// SIMATIC S7-200 project (STEP 7-Micro/WIN), CPU 224XP CN REL 02.01

ORGANIZATION_BLOCK 主程序:OB1
TITLE=程序注释；自由口通讯（甲机通过自由口通讯控制乙机电机）
BEGIN
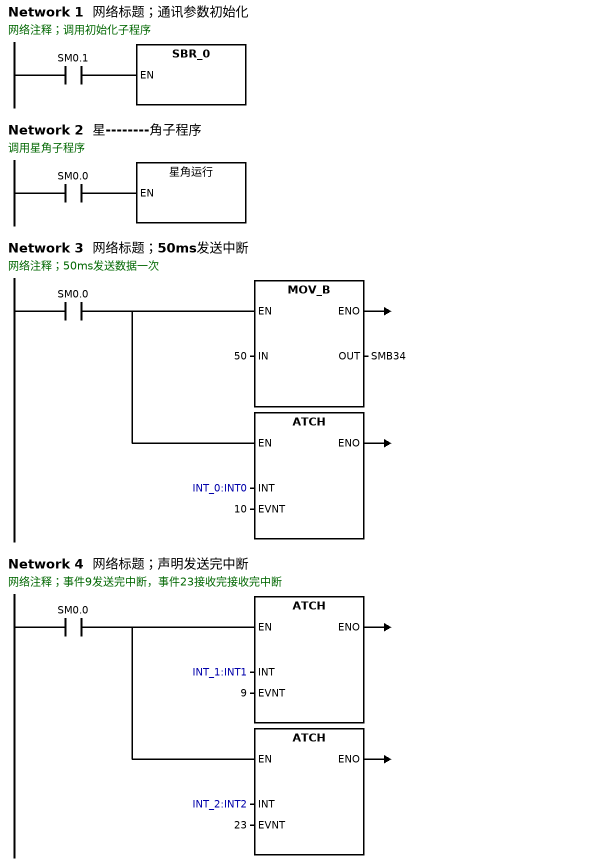
Network 1 // 网络标题；通讯参数初始化
// 网络注释；调用初始化子程序
// (network saved uncompiled; LAD cells follow)
// row 0: c0 -| |- SM0.1  c1 [SBR_0 EN:=power@row0]
Network 2 // 星--------角子程序
// 调用星角子程序
// (network saved uncompiled; LAD cells follow)
// row 0: c0 -| |- SM0.0  c1 [星角运行 EN:=power@row0]
Network 3 // 网络标题；50ms发送中断
// 网络注释；50ms发送数据一次
LD     SM0.0
MOVB   50, SMB34
ATCH   INT_0:INT0, 10
Network 4 // 网络标题；声明发送完中断
// 网络注释；事件9发送完中断，事件23接收完接收完中断
LD     SM0.0
ATCH   INT_1:INT1, 9
ATCH   INT_2:INT2, 23
END_ORGANIZATION_BLOCK

SUBROUTINE_BLOCK SBR_0:SBR0
TITLE=子程序注释：初始化通讯参数
BEGIN
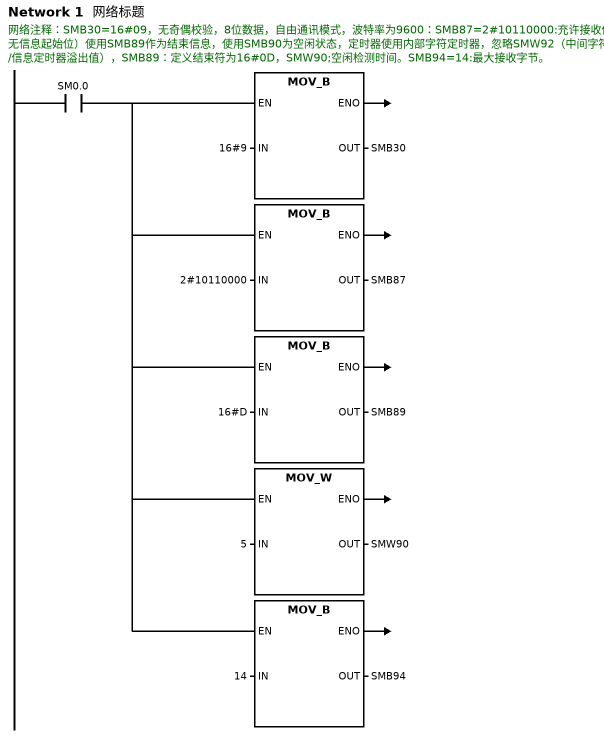
Network 1 // 网络标题
// 网络注释：SMB30=16#09，无奇偶校验，8位数据，自由通讯模式，波特率为9600：SMB87=2#10110000:充许接收信息，忽略SMB88(无信息起始位）使用SMB89作为结束信息，使用SMB90为空闲状态，定时器使用内部字符定时器，忽略SMW92（中间字符 /信息定时器溢出值），SMB89：定义结束符为16#0D，SMW90;空闲检测时间。SMB94=14:最大接收字节。
LD     SM0.0
MOVB   16#9, SMB30
MOVB   2#10110000, SMB87
MOVB   16#D, SMB89
MOVW   5, SMW90
MOVB   14, SMB94
END_SUBROUTINE_BLOCK

SUBROUTINE_BLOCK 星角运行:SBR1
TITLE=子程序注释
BEGIN
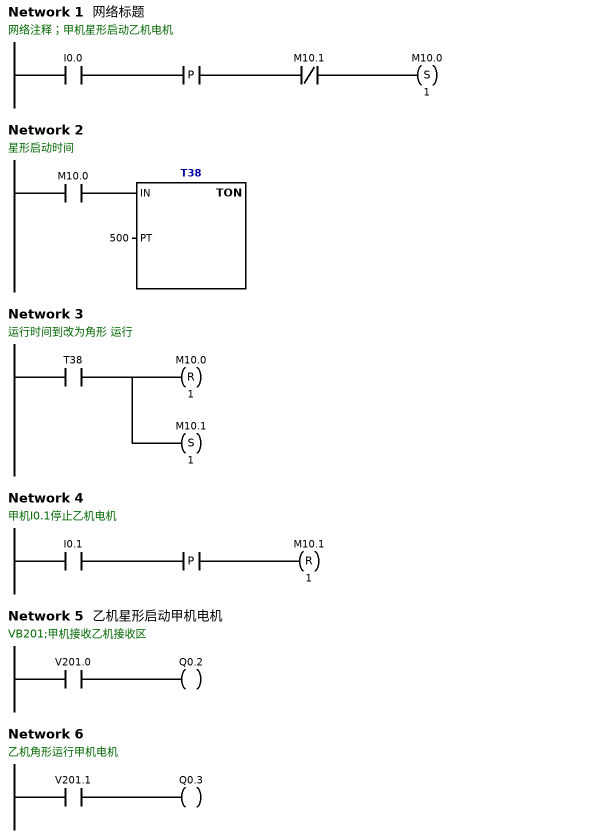
Network 1 // 网络标题
// 网络注释；甲机星形启动乙机电机
// (network saved uncompiled; LAD cells follow)
// row 0: c0 -| |- I0.0  c1 -|P|-  c2 -|/|- M10.1  c3 -(S) M10.0, 1
Network 2
// 星形启动时间
// (network saved uncompiled; LAD cells follow)
// row 0: c0 -| |- M10.0  c1 [TON T38 IN:=power@row0, PT:=500]
// row 1: c1 [box]
Network 3
// 运行时间到改为角形 运行
// (network saved uncompiled; LAD cells follow)
// row 0: c0 -| |- T38 v  c1 -(R) M10.0, 1
// row 1: c0 ^  c1 -(S) M10.1, 1
Network 4
// 甲机I0.1停止乙机电机
// (network saved uncompiled; LAD cells follow)
// row 0: c0 -| |- I0.1  c1 -|P|-  c2 -(R) M10.1, 1
Network 5 // 乙机星形启动甲机电机
// VB201;甲机接收乙机接收区
// (network saved uncompiled; LAD cells follow)
// row 0: c0 -| |- V201.0  c1 -( ) Q0.2
Network 6
// 乙机角形运行甲机电机
// (network saved uncompiled; LAD cells follow)
// row 0: c0 -| |- V201.1  c1 -( ) Q0.3
END_SUBROUTINE_BLOCK

INTERRUPT_BLOCK INT_0:INT0
TITLE=50ms间隔发送中断程序
BEGIN
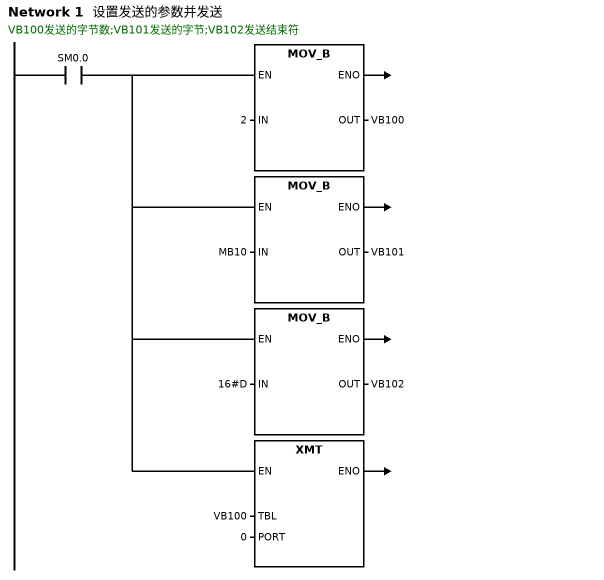
Network 1 // 设置发送的参数并发送
// VB100发送的字节数;VB101发送的字节;VB102发送结束符
LD     SM0.0
MOVB   2, VB100
MOVB   MB10, VB101
MOVB   16#D, VB102
XMT    VB100, 0
END_INTERRUPT_BLOCK

INTERRUPT_BLOCK INT_1:INT1
TITLE=数据发送完后执行此中断程序
BEGIN
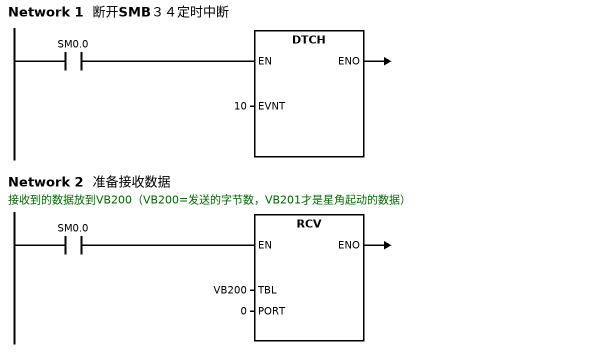
Network 1 // 断开SMB３４定时中断
LD     SM0.0
DTCH   10
Network 2 // 准备接收数据
// 接收到的数据放到VB200（VB200=发送的字节数，VB201才是星角起动的数据）
LD     SM0.0
RCV    VB200, 0
END_INTERRUPT_BLOCK

INTERRUPT_BLOCK INT_2:INT2
TITLE=
BEGIN
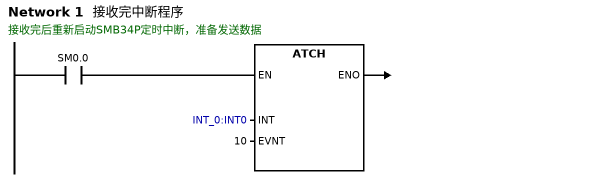
Network 1 // 接收完中断程序
// 接收完后重新启动SMB34P定时中断，准备发送数据
LD     SM0.0
ATCH   INT_0:INT0, 10
END_INTERRUPT_BLOCK
